(* Logix 5000 project; controller NSH_PLC1 vendor 1 type 14 code 167 rev 32.11; software revision 32.02; part 8 of 12 *)
(* tags used below, declared in another part *)
   CTR_HornBeeps : COUNTER;   // Number of times horn beeps
   FaultPresent : BOOL;   // A Huller-Sheller Fault is Present
   FaultReset : BOOL;   // Huller-Sheller Fault Reset
   HS_AlarmPulseHorn : BOOL;   // Huller Sheller, New Alarm, Pulse Horn
   HS_FaultResetHorn : BOOL;   // Hullwe Sheller, Fault Reset, sound Horn
   NewFault : BOOL;   // New Huller-Sheller Fault has just occured
   NewFaultBeepHorn : BOOL;   // NewFault or Warning, Pulse Horn
   NewWarning : BOOL;   // New Huller-Sheller Warning has just occured
   Num_Faults : DINT;   // Number of Huller-Sheller Faults
   Num_Faults_LS : DINT;   // Number of Huller-Sheller Faults Last PLC Scan
   Num_Warning_LS : DINT;   // Number of Huller-Sheller Warnings Last Scan, Detect New
   Num_Warnings : DINT;   // Number of Huller-Sheller Warnings
   TempMotor : Motor;   // Temp Motor Tag for Subroutines
   TMR_HornFlasher : TIMER;   // Fault Horn Flasher timer
   TMR_HS_FaultResetHorn : TIMER;   // Huller Sheller, Fault Reset, sound Horn
   C10 : Motor;   // Auger
   C8 : Motor;   // Auger
   C9 : Motor;   // Auger
   CL1 : Motor;   // Auger
   CL2 : Motor;   // Auger
   CL3 : Motor;   // Auger
   CL4 : Motor;   // Auger
   CL5 : Motor;   // Auger
   CL6 : Motor;   // Auger
   CR_RunHS : BOOL;   // Run Hullers & Shellers Relay
   D11 : Motor;   // Auger
   D12 : Motor;   // Auger
   D13 : Motor;   // Auger
   D14 : Motor;   // Auger
   DL1 : Motor;   // Auger
   H1 : Motor;   // Conv.
   H10 : Motor;   // Auger
   H11 : Motor;   // Ele.
   H12 : Motor;   // Auger
   H13 : Motor;   // Auger
   H14A : Motor;   // Shr. Roll
   H14B : Motor;   // Shr. Roll
   H14C : Motor;   // Vib.
   H15A : Motor;   // Aspirator
   H15B : Motor;   // Aspirator
   H16 : Motor;   // Auger
   H17 : Motor;   // Roll Fd.
   H18A : Motor;   // Shr. Roll
   H18B : Motor;   // Shr. Roll
   H18C : Motor;   // Vib.
   H19A : Motor;   // Aspirator
   H19B : Motor;   // Aspirator
   H20A : Motor;   // Shr. Roll
   H20B : Motor;   // Shr. Roll
   H20C : Motor;   // Vib.
   H21A : Motor;   // Aspirator
   H21B : Motor;   // Aspirator
   H22 : Motor;   // BMM
   H23A : Motor;   // Aspirator
   H23B : Motor;   // Aspirator
   H24A : Motor;   // Aspirator
   H24B : Motor;   // Aspirator
   H25 : Motor;   // Ele.
   H26 : Motor;   // Auger
   H27 : Motor;   // Auger
   H28A : Motor;   // HC Vib.
   H28B : Motor;   // Hard Crkr.
   H28C : Motor;   // S.Roll
   H28D : Motor;   // Shr.Roll.
   H29A : Motor;   // Aspirator
   H29B : Motor;   // Aspirator
   H30 : Motor;   // Auger
   H31 : Motor;   // Roll Fdr.
   H32A : Motor;   // HS Cracker
   H32B : Motor;   // Hard Crkr.
   H32C : Motor;   // Shr.Roll.
   H33B : Motor;   // Aspirator
   H36 : Motor;   // BMM
   H37A : Motor;   // Aspirator
   H37B : Motor;   // Aspirator
   H38A : Motor;   // Aspirator
   H38B : Motor;   // Aspirator
   H39 : Motor;   // Ele.
   H3A : Motor;   // Incline
   H3B : Motor;   // Ele.
   H4 : Motor;   // Auger
   H40 : Motor;   // Auger
   H41 : Motor;   // Auger
   H46 : Motor;   // BMM
   H47A : Motor;   // Aspirator
   H47B : Motor;   // Aspirator
   H48A : Motor;   // Aspirator
   H48B : Motor;   // Aspirator
   H5 : Motor;   // Auger
   H6 : Motor;   // Roll Fd.
   H7 : Motor;   // BMM
   H8A : Motor;   // Aspirator
   H8B : Motor;   // Aspirator
   H9A : Motor;   // Aspirator
   H9B : Motor;   // Aspirator
   LS101 : BOOL;   // Dummy Limit Switch
   M16R : Motor;   // Conveyor
   MainBin1 : MainBins;   // PreClean to Huller, Main Bin #1
   MainBin2 : MainBins;   // PreClean to Huller, Main Bin #1
   MainBin3 : MainBins;   // PreClean to Huller, Main Bin #1
   MainBin4 : MainBins;   // PreClean to Huller, Main Bin #1
   MainBin5 : MainBins;   // PreClean to Huller, Main Bin #1
   MainBin6 : MainBins;   // PreClean to Huller, Main Bin #1
   MainBin7 : MainBins;   // PreClean to Huller, Main Bin #1
   MainBin8 : MainBins;   // PreClean to Huller, Main Bin #1
   PB_HSFaultReset : BOOL;   // Huller Sheller, Fault Reset Button
   PBL_PCFaultReset : BOOL;   // PreClean Fault Reset Button Light
   S47 : Motor;   // Auger
   S48 : Motor;   // Auger
   S49 : Motor;   // Auger
   S50 : Motor;   // Auger
   SL1 : Motor;   // Auger
(* HullerSheller, continued *)

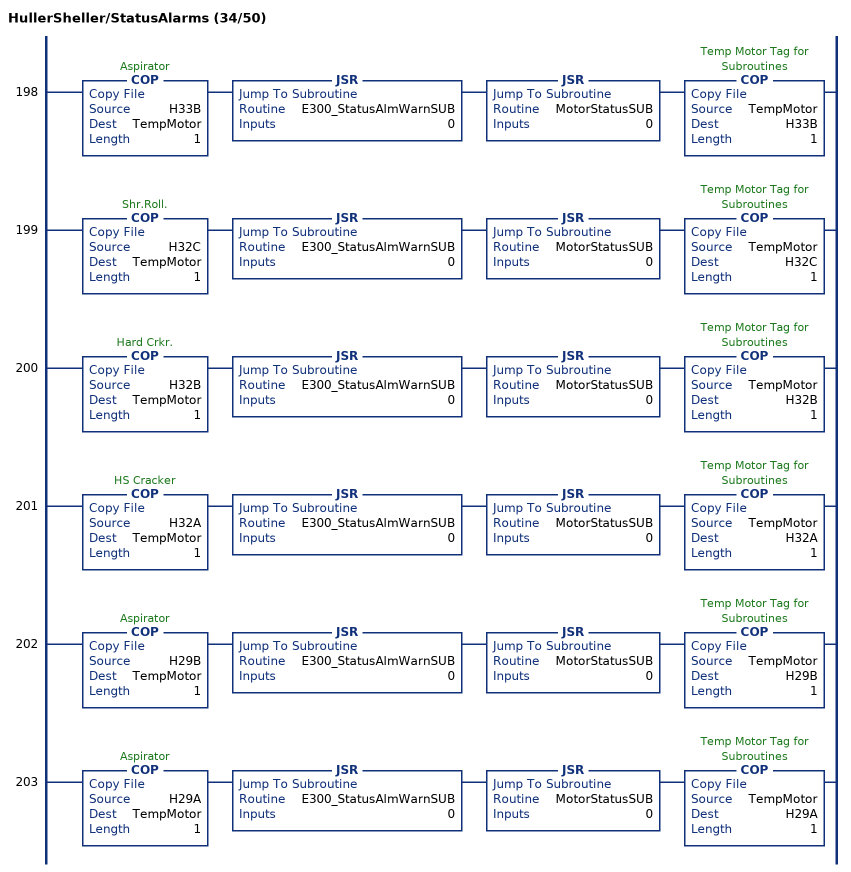
   [picture p162: HullerSheller/StatusAlarms rungs 198-203]
   198: COP(H33B,TempMotor,1)JSR(E300_StatusAlmWarnSUB,0)JSR(MotorStatusSUB,0)COP(TempMotor,H33B,1);
   199: COP(H32C,TempMotor,1)JSR(E300_StatusAlmWarnSUB,0)JSR(MotorStatusSUB,0)COP(TempMotor,H32C,1);
   200: COP(H32B,TempMotor,1)JSR(E300_StatusAlmWarnSUB,0)JSR(MotorStatusSUB,0)COP(TempMotor,H32B,1);
   201: COP(H32A,TempMotor,1)JSR(E300_StatusAlmWarnSUB,0)JSR(MotorStatusSUB,0)COP(TempMotor,H32A,1);
   202: COP(H29B,TempMotor,1)JSR(E300_StatusAlmWarnSUB,0)JSR(MotorStatusSUB,0)COP(TempMotor,H29B,1);
   203: COP(H29A,TempMotor,1)JSR(E300_StatusAlmWarnSUB,0)JSR(MotorStatusSUB,0)COP(TempMotor,H29A,1);
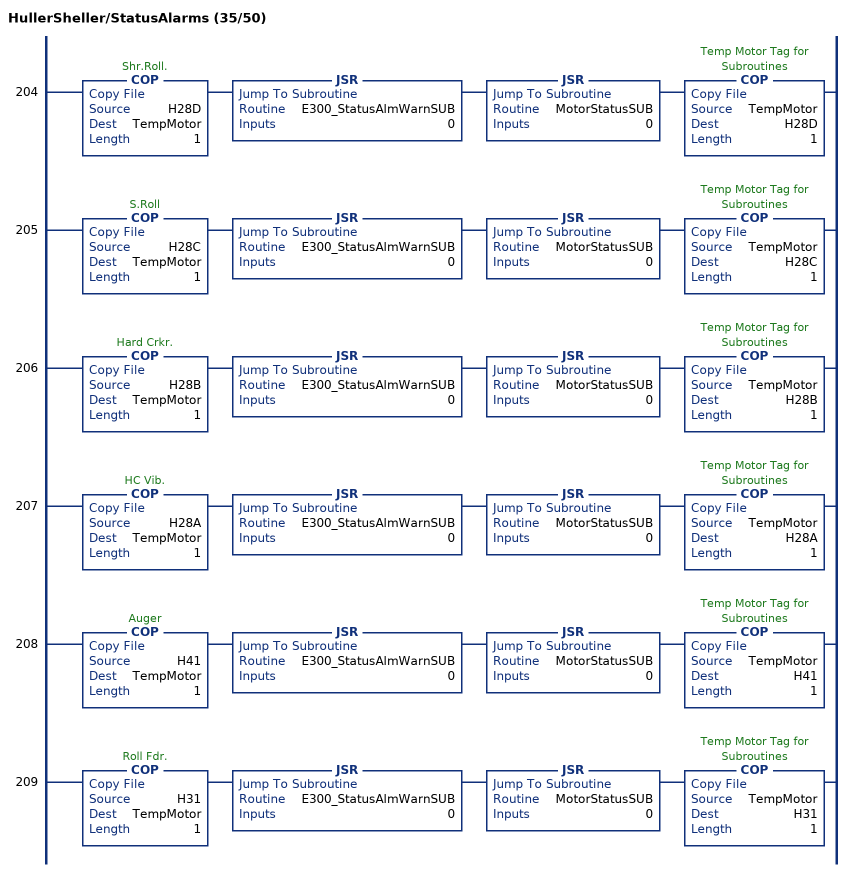
   204: COP(H28D,TempMotor,1)JSR(E300_StatusAlmWarnSUB,0)JSR(MotorStatusSUB,0)COP(TempMotor,H28D,1);
   205: COP(H28C,TempMotor,1)JSR(E300_StatusAlmWarnSUB,0)JSR(MotorStatusSUB,0)COP(TempMotor,H28C,1);
   206: COP(H28B,TempMotor,1)JSR(E300_StatusAlmWarnSUB,0)JSR(MotorStatusSUB,0)COP(TempMotor,H28B,1);
   207: COP(H28A,TempMotor,1)JSR(E300_StatusAlmWarnSUB,0)JSR(MotorStatusSUB,0)COP(TempMotor,H28A,1);
   208: COP(H41,TempMotor,1)JSR(E300_StatusAlmWarnSUB,0)JSR(MotorStatusSUB,0)COP(TempMotor,H41,1);
   209: COP(H31,TempMotor,1)JSR(E300_StatusAlmWarnSUB,0)JSR(MotorStatusSUB,0)COP(TempMotor,H31,1);
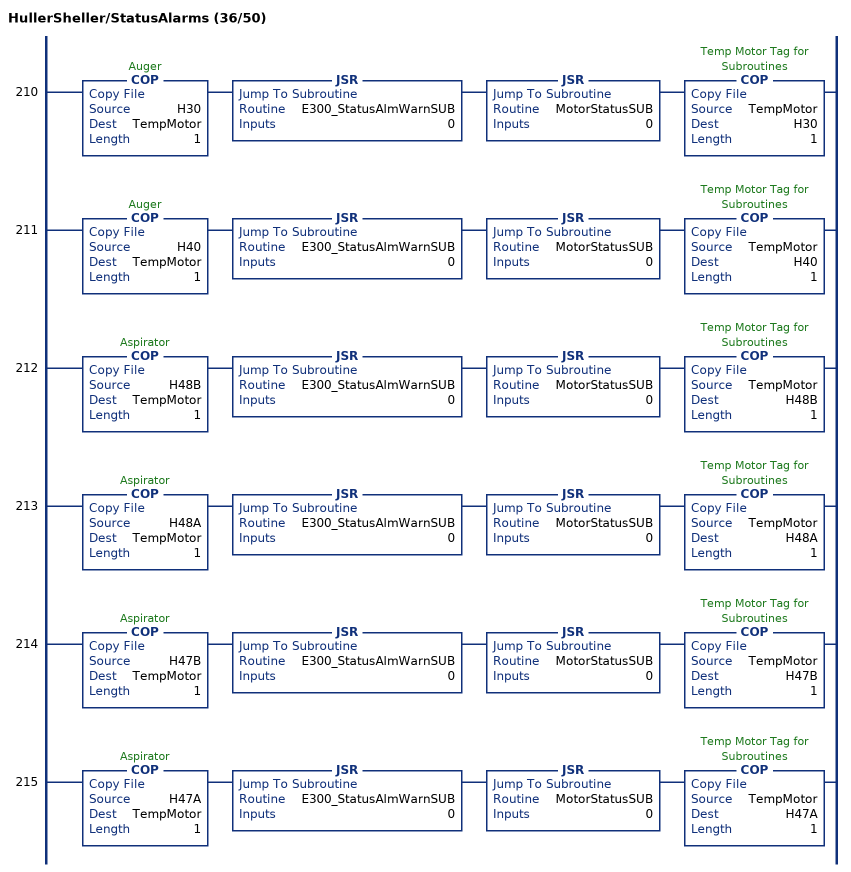
   210: COP(H30,TempMotor,1)JSR(E300_StatusAlmWarnSUB,0)JSR(MotorStatusSUB,0)COP(TempMotor,H30,1);
   211: COP(H40,TempMotor,1)JSR(E300_StatusAlmWarnSUB,0)JSR(MotorStatusSUB,0)COP(TempMotor,H40,1);
   212: COP(H48B,TempMotor,1)JSR(E300_StatusAlmWarnSUB,0)JSR(MotorStatusSUB,0)COP(TempMotor,H48B,1);
   213: COP(H48A,TempMotor,1)JSR(E300_StatusAlmWarnSUB,0)JSR(MotorStatusSUB,0)COP(TempMotor,H48A,1);
   214: COP(H47B,TempMotor,1)JSR(E300_StatusAlmWarnSUB,0)JSR(MotorStatusSUB,0)COP(TempMotor,H47B,1);
   215: COP(H47A,TempMotor,1)JSR(E300_StatusAlmWarnSUB,0)JSR(MotorStatusSUB,0)COP(TempMotor,H47A,1);
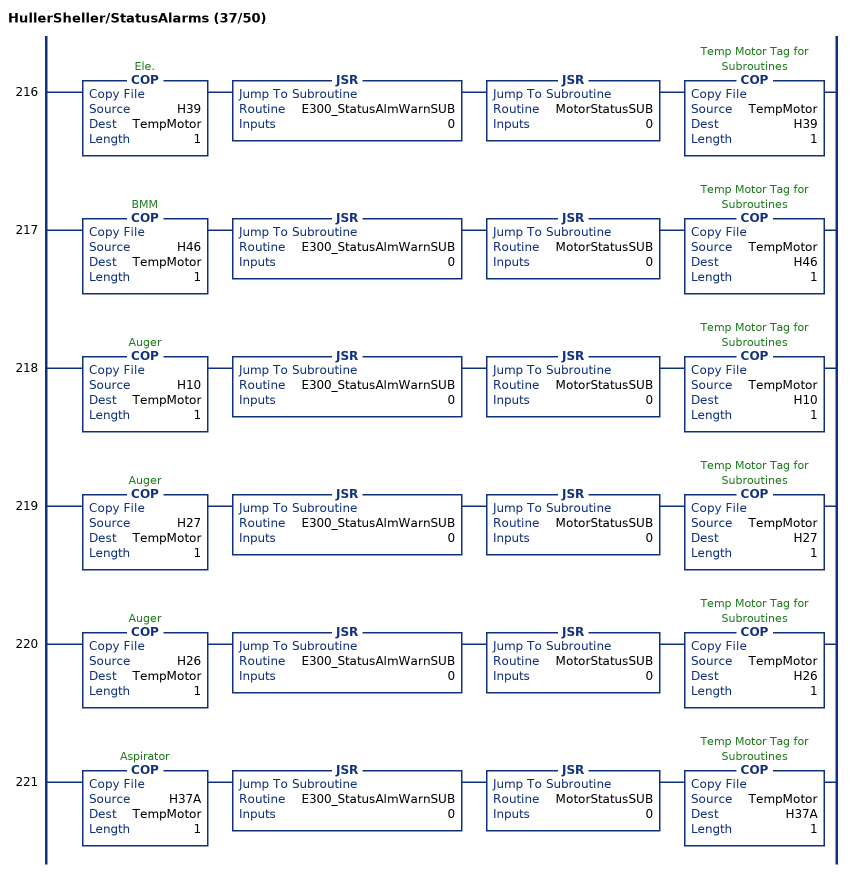
   216: COP(H39,TempMotor,1)JSR(E300_StatusAlmWarnSUB,0)JSR(MotorStatusSUB,0)COP(TempMotor,H39,1);
   217: COP(H46,TempMotor,1)JSR(E300_StatusAlmWarnSUB,0)JSR(MotorStatusSUB,0)COP(TempMotor,H46,1);
   218: COP(H10,TempMotor,1)JSR(E300_StatusAlmWarnSUB,0)JSR(MotorStatusSUB,0)COP(TempMotor,H10,1);
   219: COP(H27,TempMotor,1)JSR(E300_StatusAlmWarnSUB,0)JSR(MotorStatusSUB,0)COP(TempMotor,H27,1);
   220: COP(H26,TempMotor,1)JSR(E300_StatusAlmWarnSUB,0)JSR(MotorStatusSUB,0)COP(TempMotor,H26,1);
   221: COP(H37A,TempMotor,1)JSR(E300_StatusAlmWarnSUB,0)JSR(MotorStatusSUB,0)COP(TempMotor,H37A,1);
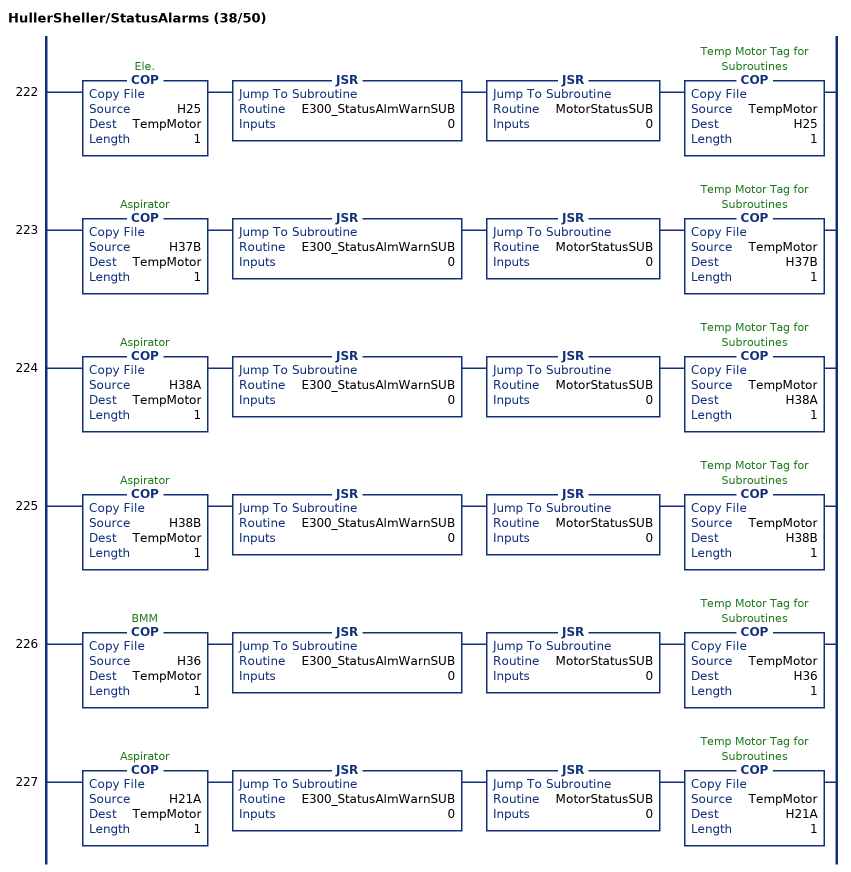
   222: COP(H25,TempMotor,1)JSR(E300_StatusAlmWarnSUB,0)JSR(MotorStatusSUB,0)COP(TempMotor,H25,1);
   223: COP(H37B,TempMotor,1)JSR(E300_StatusAlmWarnSUB,0)JSR(MotorStatusSUB,0)COP(TempMotor,H37B,1);
   224: COP(H38A,TempMotor,1)JSR(E300_StatusAlmWarnSUB,0)JSR(MotorStatusSUB,0)COP(TempMotor,H38A,1);
   225: COP(H38B,TempMotor,1)JSR(E300_StatusAlmWarnSUB,0)JSR(MotorStatusSUB,0)COP(TempMotor,H38B,1);
   226: COP(H36,TempMotor,1)JSR(E300_StatusAlmWarnSUB,0)JSR(MotorStatusSUB,0)COP(TempMotor,H36,1);
   227: COP(H21A,TempMotor,1)JSR(E300_StatusAlmWarnSUB,0)JSR(MotorStatusSUB,0)COP(TempMotor,H21A,1);
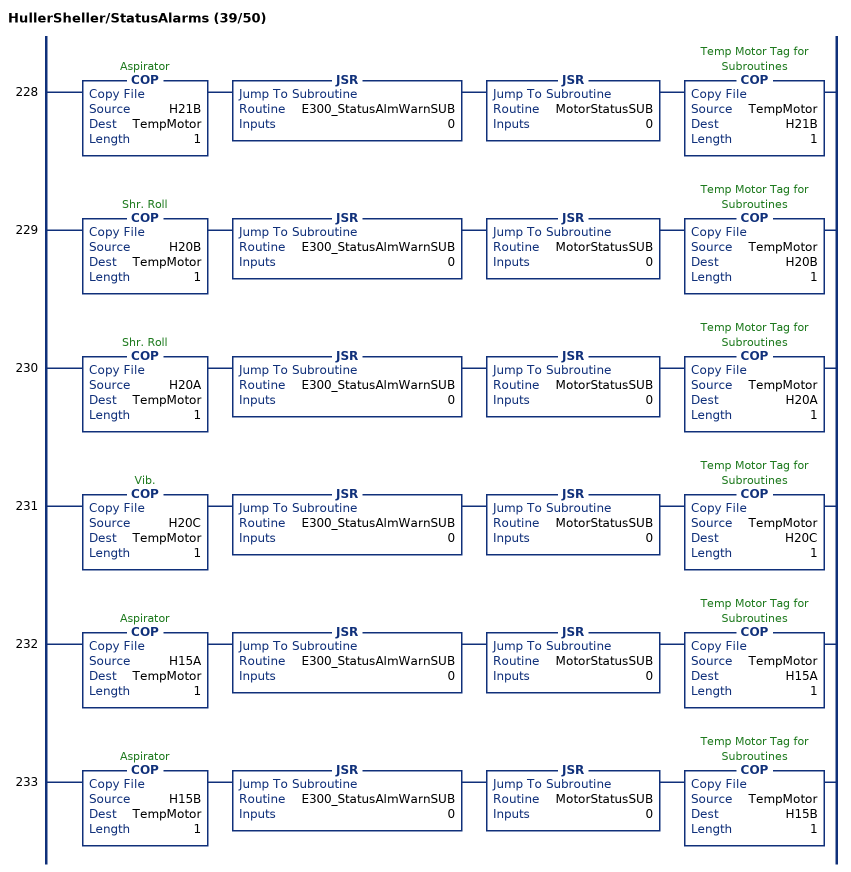
   228: COP(H21B,TempMotor,1)JSR(E300_StatusAlmWarnSUB,0)JSR(MotorStatusSUB,0)COP(TempMotor,H21B,1);
   229: COP(H20B,TempMotor,1)JSR(E300_StatusAlmWarnSUB,0)JSR(MotorStatusSUB,0)COP(TempMotor,H20B,1);
   230: COP(H20A,TempMotor,1)JSR(E300_StatusAlmWarnSUB,0)JSR(MotorStatusSUB,0)COP(TempMotor,H20A,1);
   231: COP(H20C,TempMotor,1)JSR(E300_StatusAlmWarnSUB,0)JSR(MotorStatusSUB,0)COP(TempMotor,H20C,1);
   232: COP(H15A,TempMotor,1)JSR(E300_StatusAlmWarnSUB,0)JSR(MotorStatusSUB,0)COP(TempMotor,H15A,1);
   233: COP(H15B,TempMotor,1)JSR(E300_StatusAlmWarnSUB,0)JSR(MotorStatusSUB,0)COP(TempMotor,H15B,1);
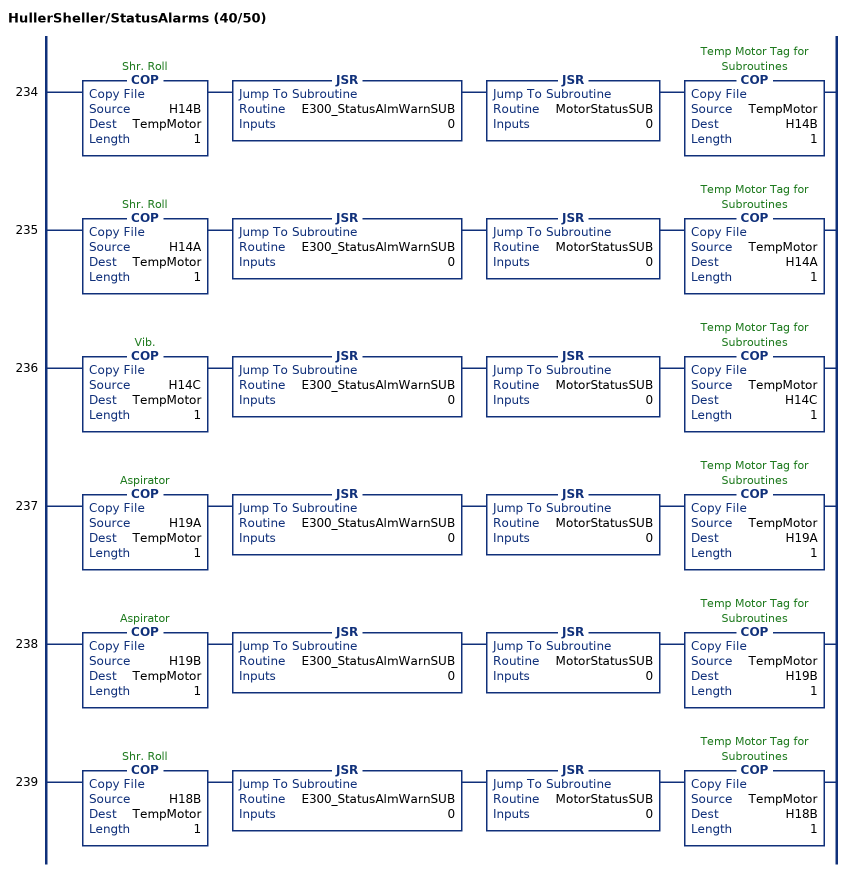
   234: COP(H14B,TempMotor,1)JSR(E300_StatusAlmWarnSUB,0)JSR(MotorStatusSUB,0)COP(TempMotor,H14B,1);
   235: COP(H14A,TempMotor,1)JSR(E300_StatusAlmWarnSUB,0)JSR(MotorStatusSUB,0)COP(TempMotor,H14A,1);
   236: COP(H14C,TempMotor,1)JSR(E300_StatusAlmWarnSUB,0)JSR(MotorStatusSUB,0)COP(TempMotor,H14C,1);
   237: COP(H19A,TempMotor,1)JSR(E300_StatusAlmWarnSUB,0)JSR(MotorStatusSUB,0)COP(TempMotor,H19A,1);
   238: COP(H19B,TempMotor,1)JSR(E300_StatusAlmWarnSUB,0)JSR(MotorStatusSUB,0)COP(TempMotor,H19B,1);
   239: COP(H18B,TempMotor,1)JSR(E300_StatusAlmWarnSUB,0)JSR(MotorStatusSUB,0)COP(TempMotor,H18B,1);
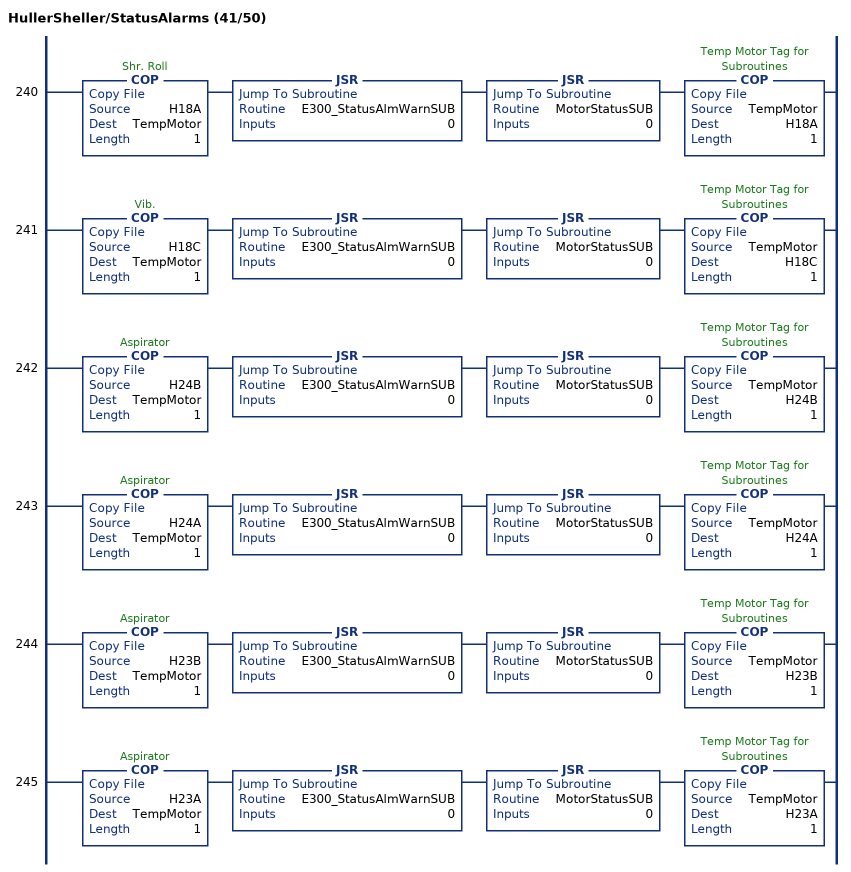
   240: COP(H18A,TempMotor,1)JSR(E300_StatusAlmWarnSUB,0)JSR(MotorStatusSUB,0)COP(TempMotor,H18A,1);
   241: COP(H18C,TempMotor,1)JSR(E300_StatusAlmWarnSUB,0)JSR(MotorStatusSUB,0)COP(TempMotor,H18C,1);
   242: COP(H24B,TempMotor,1)JSR(E300_StatusAlmWarnSUB,0)JSR(MotorStatusSUB,0)COP(TempMotor,H24B,1);
   243: COP(H24A,TempMotor,1)JSR(E300_StatusAlmWarnSUB,0)JSR(MotorStatusSUB,0)COP(TempMotor,H24A,1);
   244: COP(H23B,TempMotor,1)JSR(E300_StatusAlmWarnSUB,0)JSR(MotorStatusSUB,0)COP(TempMotor,H23B,1);
   245: COP(H23A,TempMotor,1)JSR(E300_StatusAlmWarnSUB,0)JSR(MotorStatusSUB,0)COP(TempMotor,H23A,1);
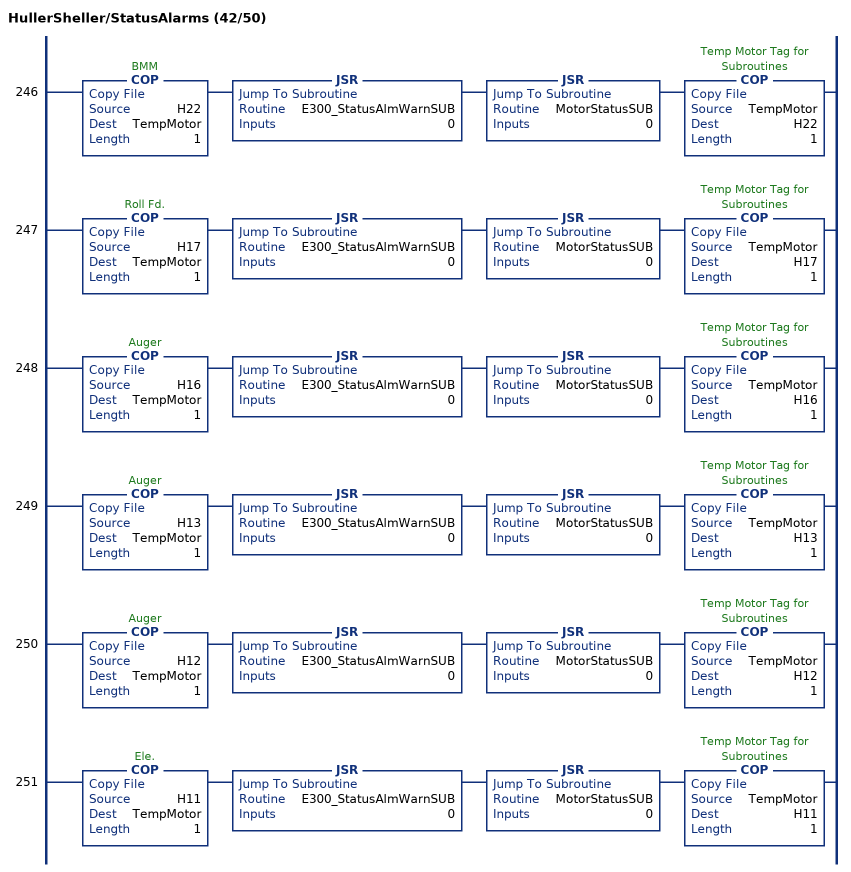
   246: COP(H22,TempMotor,1)JSR(E300_StatusAlmWarnSUB,0)JSR(MotorStatusSUB,0)COP(TempMotor,H22,1);
   247: COP(H17,TempMotor,1)JSR(E300_StatusAlmWarnSUB,0)JSR(MotorStatusSUB,0)COP(TempMotor,H17,1);
   248: COP(H16,TempMotor,1)JSR(E300_StatusAlmWarnSUB,0)JSR(MotorStatusSUB,0)COP(TempMotor,H16,1);
   249: COP(H13,TempMotor,1)JSR(E300_StatusAlmWarnSUB,0)JSR(MotorStatusSUB,0)COP(TempMotor,H13,1);
   250: COP(H12,TempMotor,1)JSR(E300_StatusAlmWarnSUB,0)JSR(MotorStatusSUB,0)COP(TempMotor,H12,1);
   251: COP(H11,TempMotor,1)JSR(E300_StatusAlmWarnSUB,0)JSR(MotorStatusSUB,0)COP(TempMotor,H11,1);
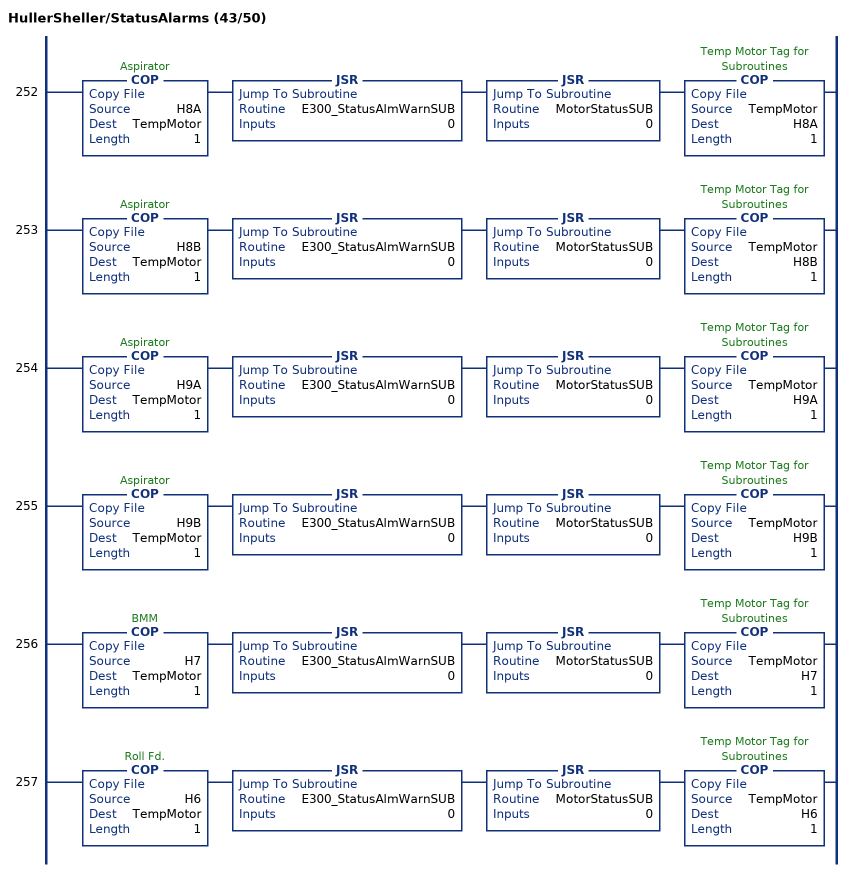
   252: COP(H8A,TempMotor,1)JSR(E300_StatusAlmWarnSUB,0)JSR(MotorStatusSUB,0)COP(TempMotor,H8A,1);
   253: COP(H8B,TempMotor,1)JSR(E300_StatusAlmWarnSUB,0)JSR(MotorStatusSUB,0)COP(TempMotor,H8B,1);
   254: COP(H9A,TempMotor,1)JSR(E300_StatusAlmWarnSUB,0)JSR(MotorStatusSUB,0)COP(TempMotor,H9A,1);
   255: COP(H9B,TempMotor,1)JSR(E300_StatusAlmWarnSUB,0)JSR(MotorStatusSUB,0)COP(TempMotor,H9B,1);
   256: COP(H7,TempMotor,1)JSR(E300_StatusAlmWarnSUB,0)JSR(MotorStatusSUB,0)COP(TempMotor,H7,1);
   257: COP(H6,TempMotor,1)JSR(E300_StatusAlmWarnSUB,0)JSR(MotorStatusSUB,0)COP(TempMotor,H6,1);
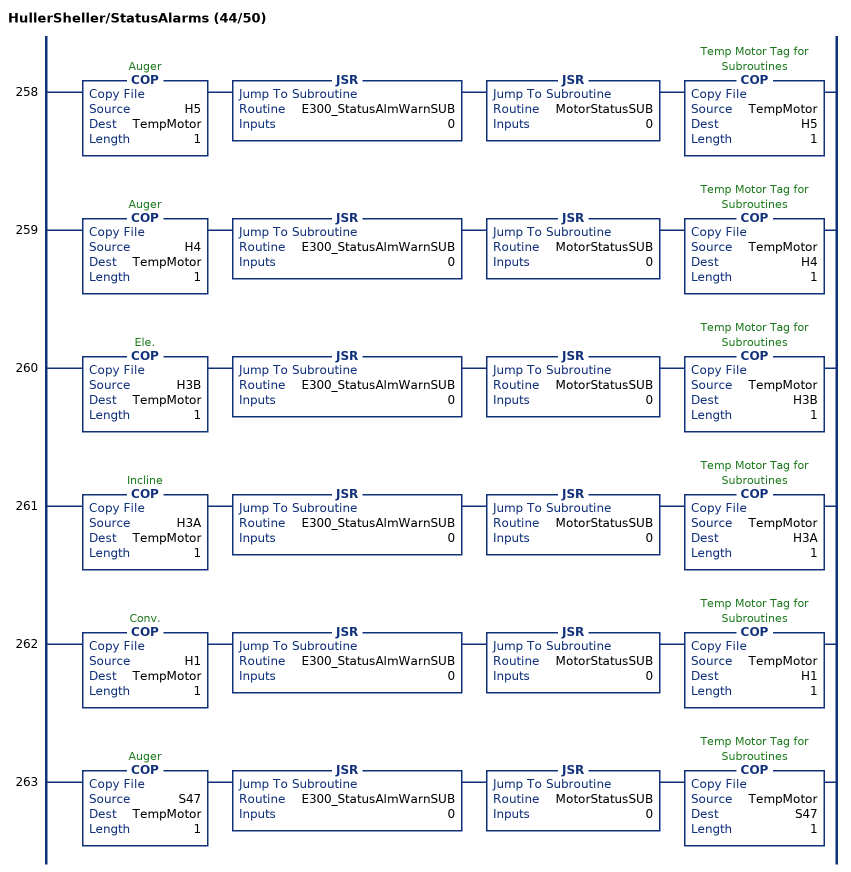
   258: COP(H5,TempMotor,1)JSR(E300_StatusAlmWarnSUB,0)JSR(MotorStatusSUB,0)COP(TempMotor,H5,1);
   259: COP(H4,TempMotor,1)JSR(E300_StatusAlmWarnSUB,0)JSR(MotorStatusSUB,0)COP(TempMotor,H4,1);
   260: COP(H3B,TempMotor,1)JSR(E300_StatusAlmWarnSUB,0)JSR(MotorStatusSUB,0)COP(TempMotor,H3B,1);
   261: COP(H3A,TempMotor,1)JSR(E300_StatusAlmWarnSUB,0)JSR(MotorStatusSUB,0)COP(TempMotor,H3A,1);
   262: COP(H1,TempMotor,1)JSR(E300_StatusAlmWarnSUB,0)JSR(MotorStatusSUB,0)COP(TempMotor,H1,1);
   263: COP(S47,TempMotor,1)JSR(E300_StatusAlmWarnSUB,0)JSR(MotorStatusSUB,0)COP(TempMotor,S47,1);
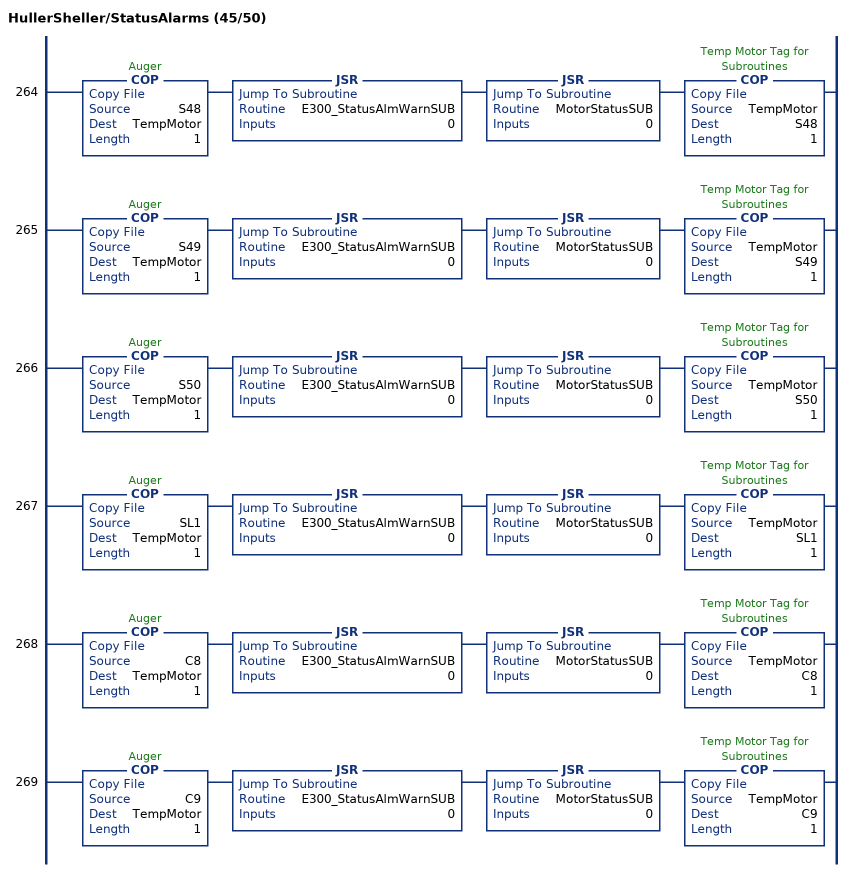
   264: COP(S48,TempMotor,1)JSR(E300_StatusAlmWarnSUB,0)JSR(MotorStatusSUB,0)COP(TempMotor,S48,1);
   265: COP(S49,TempMotor,1)JSR(E300_StatusAlmWarnSUB,0)JSR(MotorStatusSUB,0)COP(TempMotor,S49,1);
   266: COP(S50,TempMotor,1)JSR(E300_StatusAlmWarnSUB,0)JSR(MotorStatusSUB,0)COP(TempMotor,S50,1);
   267: COP(SL1,TempMotor,1)JSR(E300_StatusAlmWarnSUB,0)JSR(MotorStatusSUB,0)COP(TempMotor,SL1,1);
   268: COP(C8,TempMotor,1)JSR(E300_StatusAlmWarnSUB,0)JSR(MotorStatusSUB,0)COP(TempMotor,C8,1);
   269: COP(C9,TempMotor,1)JSR(E300_StatusAlmWarnSUB,0)JSR(MotorStatusSUB,0)COP(TempMotor,C9,1);
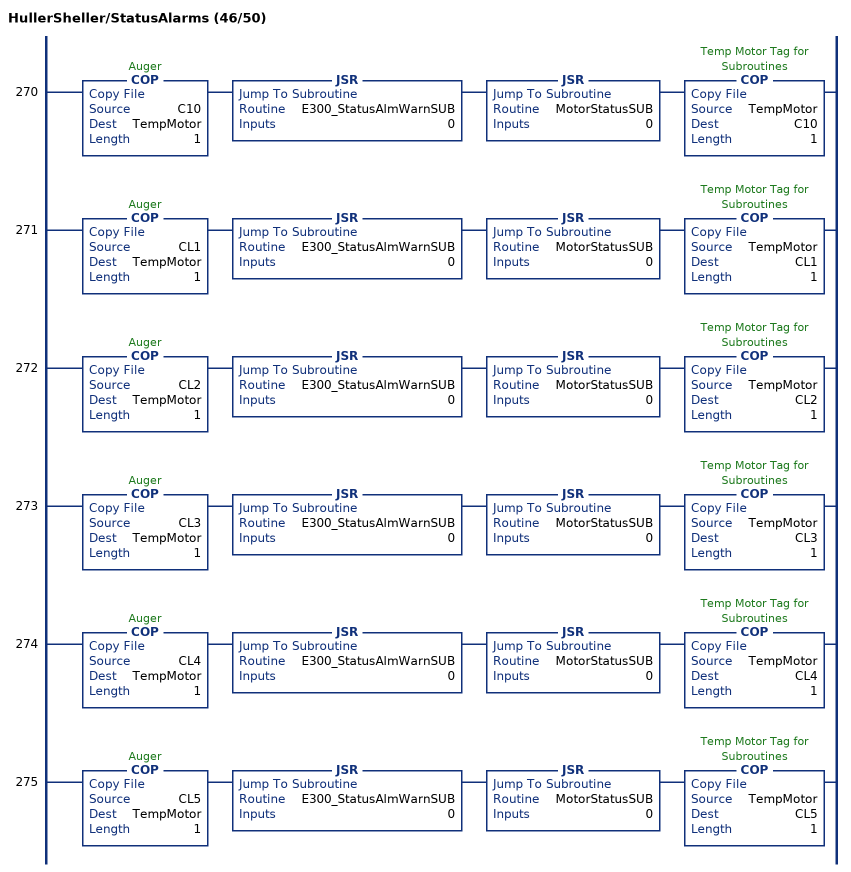
   270: COP(C10,TempMotor,1)JSR(E300_StatusAlmWarnSUB,0)JSR(MotorStatusSUB,0)COP(TempMotor,C10,1);
   271: COP(CL1,TempMotor,1)JSR(E300_StatusAlmWarnSUB,0)JSR(MotorStatusSUB,0)COP(TempMotor,CL1,1);
   272: COP(CL2,TempMotor,1)JSR(E300_StatusAlmWarnSUB,0)JSR(MotorStatusSUB,0)COP(TempMotor,CL2,1);
   273: COP(CL3,TempMotor,1)JSR(E300_StatusAlmWarnSUB,0)JSR(MotorStatusSUB,0)COP(TempMotor,CL3,1);
   274: COP(CL4,TempMotor,1)JSR(E300_StatusAlmWarnSUB,0)JSR(MotorStatusSUB,0)COP(TempMotor,CL4,1);
   275: COP(CL5,TempMotor,1)JSR(E300_StatusAlmWarnSUB,0)JSR(MotorStatusSUB,0)COP(TempMotor,CL5,1);
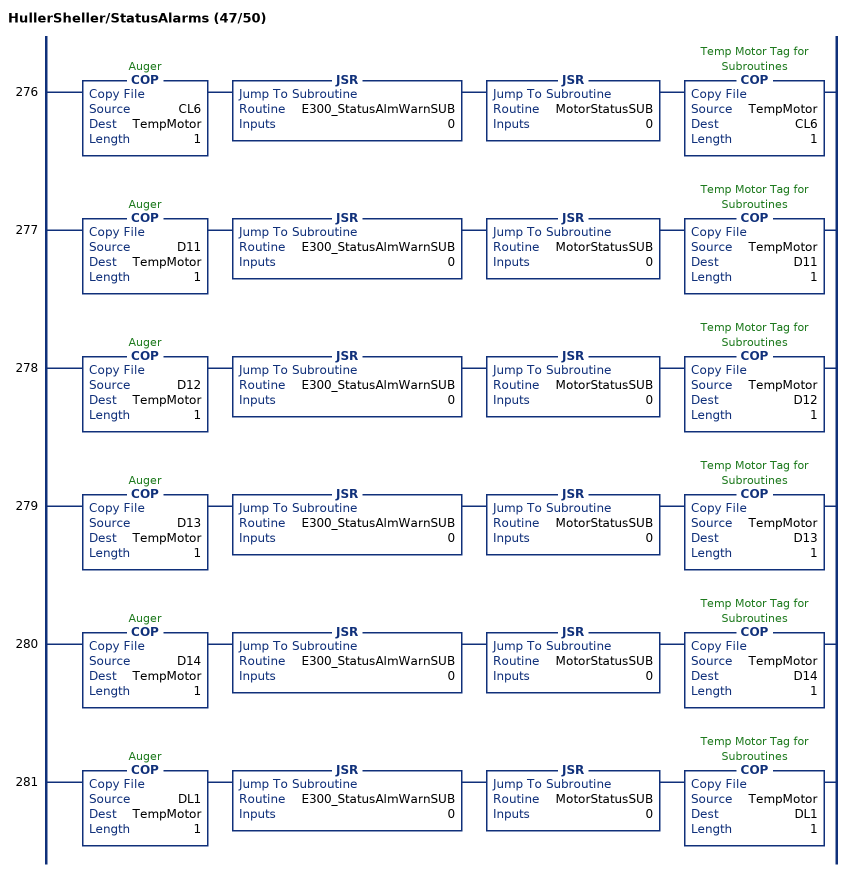
   276: COP(CL6,TempMotor,1)JSR(E300_StatusAlmWarnSUB,0)JSR(MotorStatusSUB,0)COP(TempMotor,CL6,1);
   277: COP(D11,TempMotor,1)JSR(E300_StatusAlmWarnSUB,0)JSR(MotorStatusSUB,0)COP(TempMotor,D11,1);
   278: COP(D12,TempMotor,1)JSR(E300_StatusAlmWarnSUB,0)JSR(MotorStatusSUB,0)COP(TempMotor,D12,1);
   279: COP(D13,TempMotor,1)JSR(E300_StatusAlmWarnSUB,0)JSR(MotorStatusSUB,0)COP(TempMotor,D13,1);
   280: COP(D14,TempMotor,1)JSR(E300_StatusAlmWarnSUB,0)JSR(MotorStatusSUB,0)COP(TempMotor,D14,1);
   281: COP(DL1,TempMotor,1)JSR(E300_StatusAlmWarnSUB,0)JSR(MotorStatusSUB,0)COP(TempMotor,DL1,1);
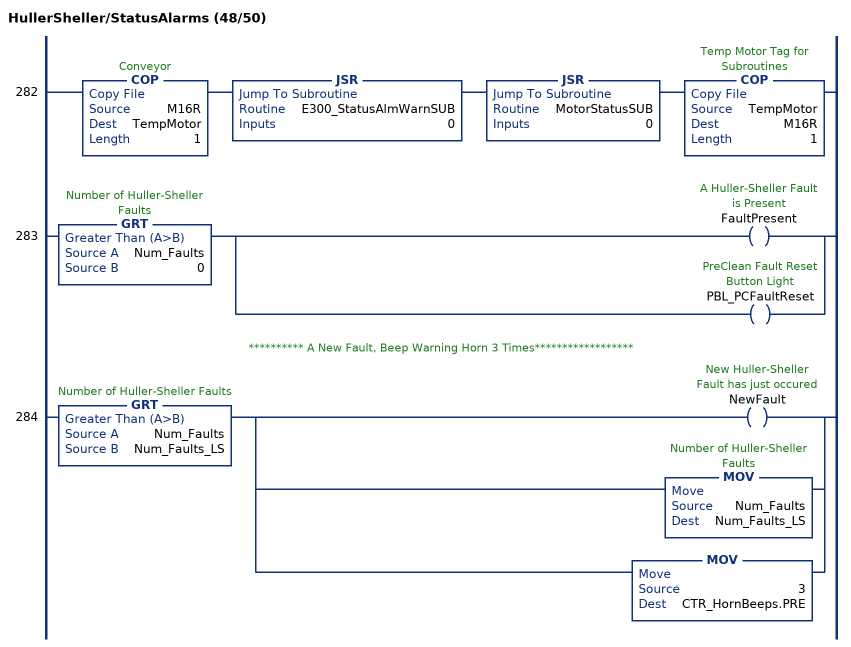
   282: COP(M16R,TempMotor,1)JSR(E300_StatusAlmWarnSUB,0)JSR(MotorStatusSUB,0)COP(TempMotor,M16R,1);
   283: GRT(Num_Faults,0)[OTE(FaultPresent) ,OTE(PBL_PCFaultReset) ];
   // ********** A New Fault, Beep Warning Horn 3 Times******************
   284: GRT(Num_Faults,Num_Faults_LS)[OTE(NewFault) ,MOV(Num_Faults,Num_Faults_LS) ,MOV(3,CTR_HornBeeps.PRE) ];
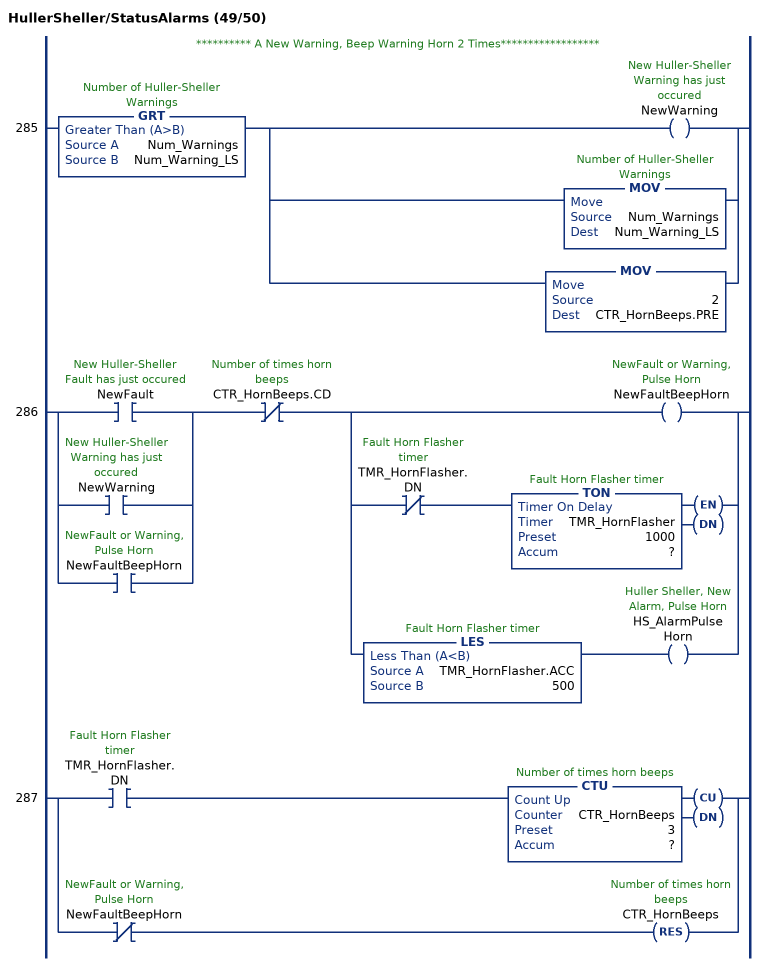
   // ********** A New Warning, Beep Warning Horn 2 Times******************
   285: GRT(Num_Warnings,Num_Warning_LS)[OTE(NewWarning) ,MOV(Num_Warnings,Num_Warning_LS) ,MOV(2,CTR_HornBeeps.PRE) ];
   286: [XIC(NewFault) ,XIC(NewWarning) ,XIC(NewFaultBeepHorn) ]XIO(CTR_HornBeeps.CD)[OTE(NewFaultBeepHorn) ,XIO(TMR_HornFlasher.DN) TON(TMR_HornFlasher,?,?) ,LES(TMR_HornFlasher.ACC,500) OTE(HS_AlarmPulseHorn) ];
   287: [XIC(TMR_HornFlasher.DN) CTU(CTR_HornBeeps,?,?) ,XIO(NewFaultBeepHorn) RES(CTR_HornBeeps) ];
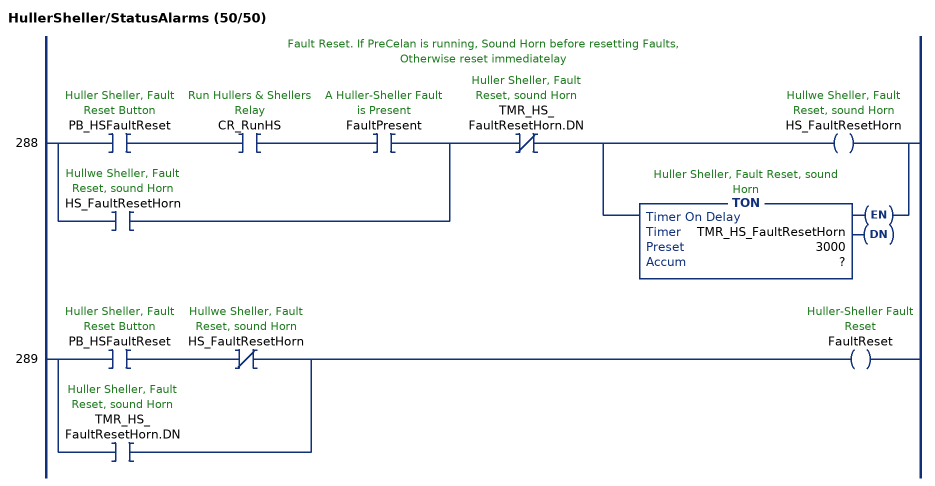
   // Fault Reset. If PreCelan is running, Sound Horn before resetting Faults,
   // Otherwise reset immediatelay
   288: [XIC(PB_HSFaultReset) XIC(CR_RunHS) XIC(FaultPresent) ,XIC(HS_FaultResetHorn) ]XIO(TMR_HS_FaultResetHorn.DN)[OTE(HS_FaultResetHorn) ,TON(TMR_HS_FaultResetHorn,?,?) ];
   289: [XIC(PB_HSFaultReset) XIO(HS_FaultResetHorn) ,XIC(TMR_HS_FaultResetHorn.DN) ]OTE(FaultReset);
END_ROUTINE
END_PROGRAM

PROGRAM Initialize   (* main routine SetRunStop_ResetHandAuto *)

ROUTINE SetRunStop_ResetHandAuto   (* ladder *)
END_ROUTINE
END_PROGRAM

PROGRAM MainProgram   (* main routine MainJSR *)

ROUTINE E300_AOP_ToMotorsSUB   (* ladder *)
// Get E300 AOP Imputs and Put Into Motor Structure
END_ROUTINE

ROUTINE Inputs_FlexIO   (* ladder *)
// Input infomation from Flex IO Inputs
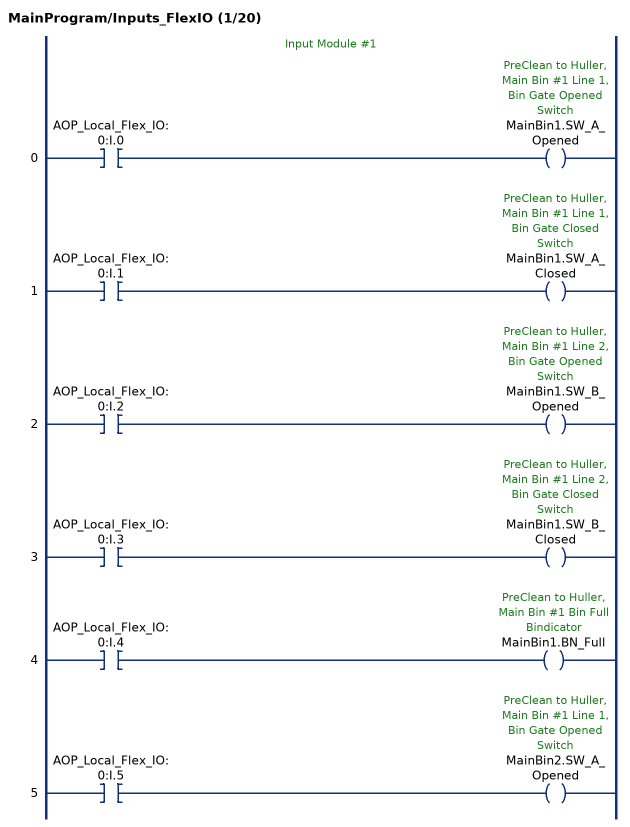
   // Input Module #1
   0: XIC(AOP_Local_Flex_IO:0:I.0)OTE(MainBin1.SW_A_Opened);
   1: XIC(AOP_Local_Flex_IO:0:I.1)OTE(MainBin1.SW_A_Closed);
   2: XIC(AOP_Local_Flex_IO:0:I.2)OTE(MainBin1.SW_B_Opened);
   3: XIC(AOP_Local_Flex_IO:0:I.3)OTE(MainBin1.SW_B_Closed);
   4: XIC(AOP_Local_Flex_IO:0:I.4)OTE(MainBin1.BN_Full);
   5: XIC(AOP_Local_Flex_IO:0:I.5)OTE(MainBin2.SW_A_Opened);
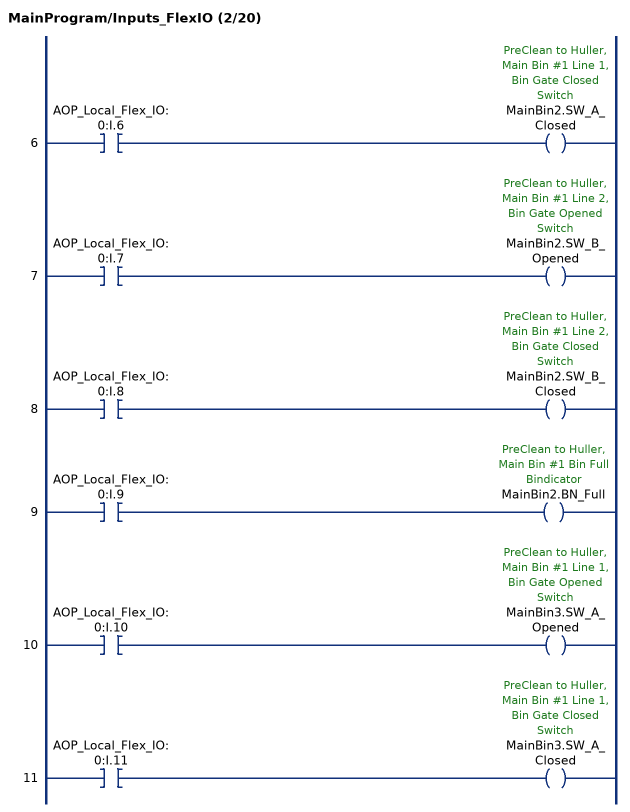
   6: XIC(AOP_Local_Flex_IO:0:I.6)OTE(MainBin2.SW_A_Closed);
   7: XIC(AOP_Local_Flex_IO:0:I.7)OTE(MainBin2.SW_B_Opened);
   8: XIC(AOP_Local_Flex_IO:0:I.8)OTE(MainBin2.SW_B_Closed);
   9: XIC(AOP_Local_Flex_IO:0:I.9)OTE(MainBin2.BN_Full);
   10: XIC(AOP_Local_Flex_IO:0:I.10)OTE(MainBin3.SW_A_Opened);
   11: XIC(AOP_Local_Flex_IO:0:I.11)OTE(MainBin3.SW_A_Closed);
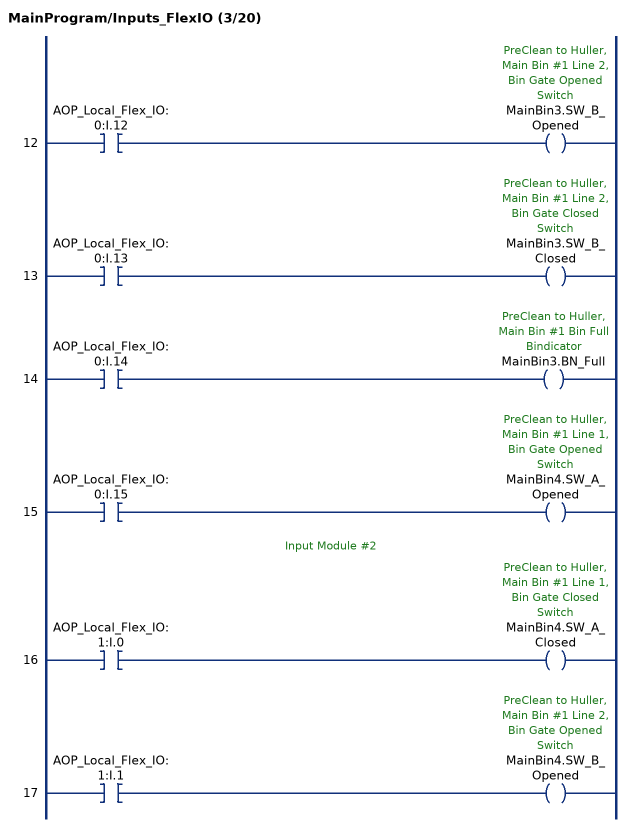
   12: XIC(AOP_Local_Flex_IO:0:I.12)OTE(MainBin3.SW_B_Opened);
   13: XIC(AOP_Local_Flex_IO:0:I.13)OTE(MainBin3.SW_B_Closed);
   14: XIC(AOP_Local_Flex_IO:0:I.14)OTE(MainBin3.BN_Full);
   15: XIC(AOP_Local_Flex_IO:0:I.15)OTE(MainBin4.SW_A_Opened);
   // Input Module #2
   16: XIC(AOP_Local_Flex_IO:1:I.0)OTE(MainBin4.SW_A_Closed);
   17: XIC(AOP_Local_Flex_IO:1:I.1)OTE(MainBin4.SW_B_Opened);
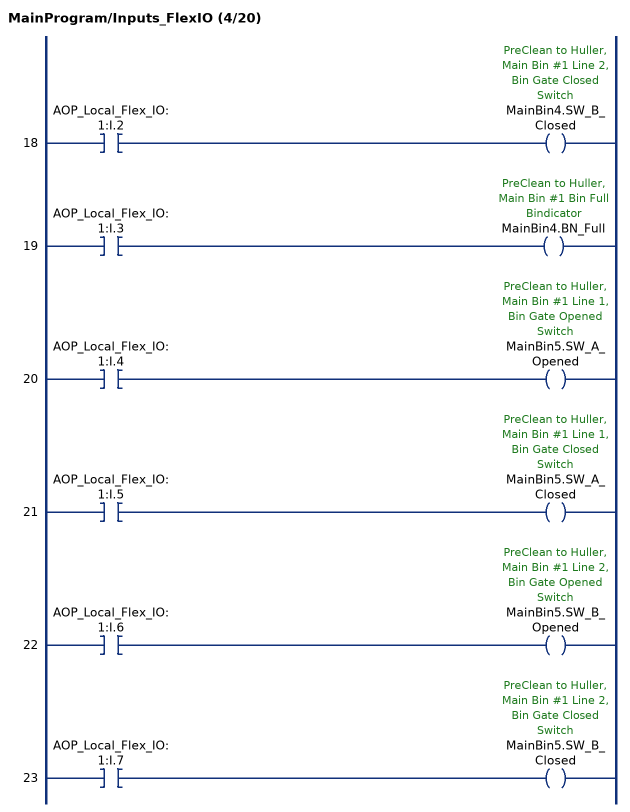
   18: XIC(AOP_Local_Flex_IO:1:I.2)OTE(MainBin4.SW_B_Closed);
   19: XIC(AOP_Local_Flex_IO:1:I.3)OTE(MainBin4.BN_Full);
   20: XIC(AOP_Local_Flex_IO:1:I.4)OTE(MainBin5.SW_A_Opened);
   21: XIC(AOP_Local_Flex_IO:1:I.5)OTE(MainBin5.SW_A_Closed);
   22: XIC(AOP_Local_Flex_IO:1:I.6)OTE(MainBin5.SW_B_Opened);
   23: XIC(AOP_Local_Flex_IO:1:I.7)OTE(MainBin5.SW_B_Closed);
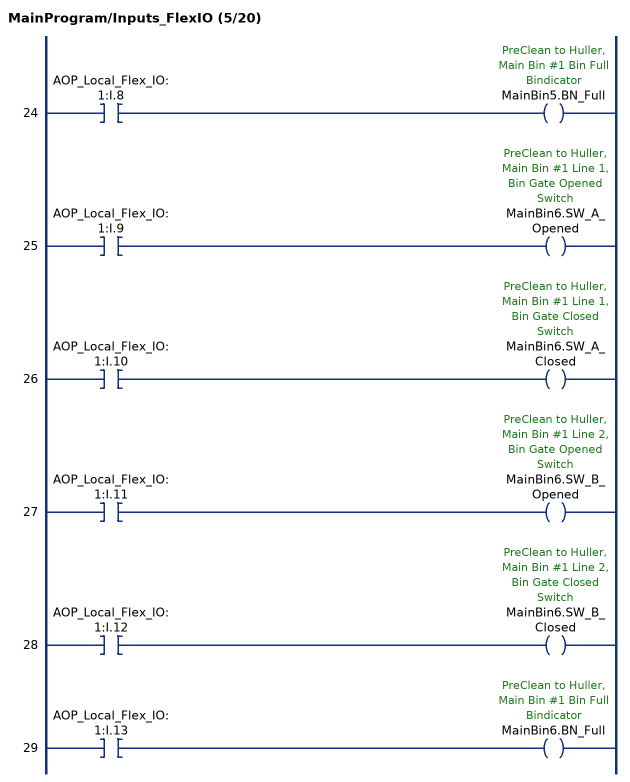
   24: XIC(AOP_Local_Flex_IO:1:I.8)OTE(MainBin5.BN_Full);
   25: XIC(AOP_Local_Flex_IO:1:I.9)OTE(MainBin6.SW_A_Opened);
   26: XIC(AOP_Local_Flex_IO:1:I.10)OTE(MainBin6.SW_A_Closed);
   27: XIC(AOP_Local_Flex_IO:1:I.11)OTE(MainBin6.SW_B_Opened);
   28: XIC(AOP_Local_Flex_IO:1:I.12)OTE(MainBin6.SW_B_Closed);
   29: XIC(AOP_Local_Flex_IO:1:I.13)OTE(MainBin6.BN_Full);
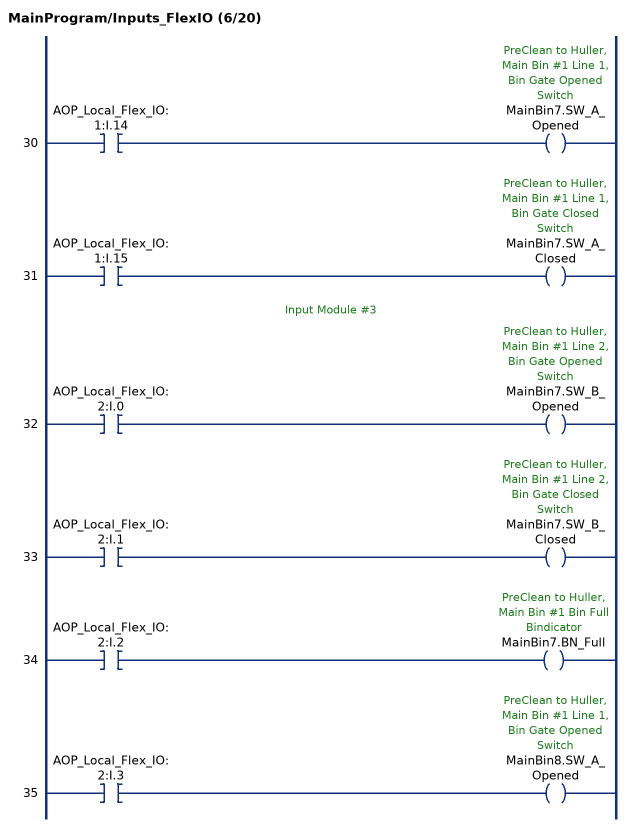
   30: XIC(AOP_Local_Flex_IO:1:I.14)OTE(MainBin7.SW_A_Opened);
   31: XIC(AOP_Local_Flex_IO:1:I.15)OTE(MainBin7.SW_A_Closed);
   // Input Module #3
   32: XIC(AOP_Local_Flex_IO:2:I.0)OTE(MainBin7.SW_B_Opened);
   33: XIC(AOP_Local_Flex_IO:2:I.1)OTE(MainBin7.SW_B_Closed);
   34: XIC(AOP_Local_Flex_IO:2:I.2)OTE(MainBin7.BN_Full);
   35: XIC(AOP_Local_Flex_IO:2:I.3)OTE(MainBin8.SW_A_Opened);
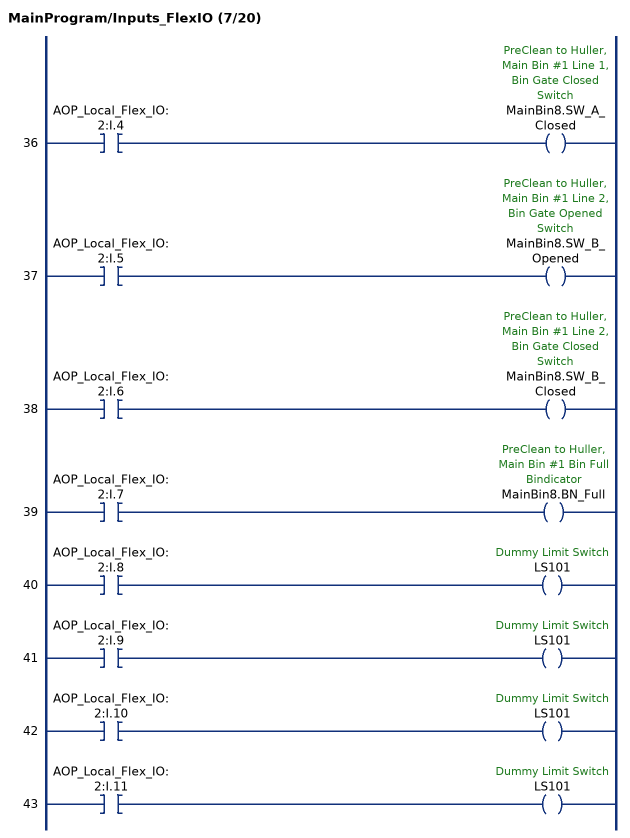
   36: XIC(AOP_Local_Flex_IO:2:I.4)OTE(MainBin8.SW_A_Closed);
   37: XIC(AOP_Local_Flex_IO:2:I.5)OTE(MainBin8.SW_B_Opened);
   38: XIC(AOP_Local_Flex_IO:2:I.6)OTE(MainBin8.SW_B_Closed);
   39: XIC(AOP_Local_Flex_IO:2:I.7)OTE(MainBin8.BN_Full);
   40: XIC(AOP_Local_Flex_IO:2:I.8)OTE(LS101);
   41: XIC(AOP_Local_Flex_IO:2:I.9)OTE(LS101);
   42: XIC(AOP_Local_Flex_IO:2:I.10)OTE(LS101);
   43: XIC(AOP_Local_Flex_IO:2:I.11)OTE(LS101);
